# EPICS substitutions: iocBoot/iocMicrotest/Microtest.substitutions
file "$(MICROTEST)/MicrotestApp/Db/Microtest.template"
{
pattern
{    P,        PORT,       ADDR}
{   Deben,   Microtest,     0}
}
